FUNCTION_BLOCK FB_FIFOTest
VAR_INPUT
END_VAR
VAR_OUTPUT
END_VAR
VAR
	fbFIFO		: FB_FIFOInt;
	
	enqTrig		: R_TRIG;
	deqTrig		: R_TRIG;
	
	bEnqueueError : BOOL;
	bDequeueError : BOOL; 
END_VAR


fbFIFO();

enqTrig(CLK := GVL_Test.bEnqueueItem);
deqTrig(CLK := GVL_Test.bDequeueItem);

IF enqTrig.Q THEN
	fbFIFO.Enqueue(i_Item := GVL_Test.itemToStored);
	bEnqueueError := fbFIFO.o_EnqueueError;
END_IF

IF deqTrig.Q THEN
	fbFIFO.Dequeue(o_Item => GVL_Test.ExportedItem);
	bDequeueError := fbFIFO.o_DequeueError;
END_IF

END_FUNCTION_BLOCK

(* stored: Version 1.1.0.1, ProductVersion 3.1.4024.2
   POU FB_FIFOTest: Id {d5fb4b37-87b6-4c80-a865-b42802c979e7}, SpecialFunc None *)
